(* --> Controller Errors <--*)
		17664	:		FC_NcErrorMsg:='Controller Errors-Parameter:"Controller ID not allowed" The value for the controller ID is not allowed,  e.g. because it has already been assigned, is less than or equal to zero, or is greater than 255.';
		17665	:		FC_NcErrorMsg:='Controller Errors-Parameter:"Controller type not allowed" The value for the controller type is unacceptable because it is not defined. Type 1: P-controller (position) . . .  Type 7: High/low speed controller  Type 8: JogStepper motor controller  Type 9: Sercos controller';
		17666	:		FC_NcErrorMsg:='Controller Errors-Parameter:"Controller operating mode not allowed" The value for the controller operating mode is not allowed.';
		17667	:		FC_NcErrorMsg:='Controller Errors-Parameter:"Weighting of the velocity pre-control not allowed" The value for the percentage weighting of the velocity pre-control is not allowed.  The parameter is pre-set to 1.0 (100%) as standard.';
		17668	:		FC_NcErrorMsg:='Controller Errors-Parameter:"Following error monitoring (position) not allowed" The value for the activation of the following error monitoring is not allowed.';
		17669	:		FC_NcErrorMsg:='Controller Errors-Parameter:"Following error (velocity) not allowed" The value for the activation of the following error monitoring (velocity) is not allowed.';
		17670	:		FC_NcErrorMsg:='Controller Errors-Parameter:"Following error window (position) not allowed" The value for the following error window (maximum allowable following error) is not allowed.';
		17671	:		FC_NcErrorMsg:='Controller Errors-Parameter:"Following error filter time (position) not allowed" The value for the following error filter time (position) is not allowed.';
		17672	:		FC_NcErrorMsg:='Controller Errors-Parameter:"Following error window (velocity) not allowed" The value for the following error window (velocity) is not allowed.';
		17673	:		FC_NcErrorMsg:='Controller Errors-Parameter:"Following error filter time (velocity) not allowed" The value for the following error filter time (velocity) is not allowed.';
		17680	:		FC_NcErrorMsg:='Controller Errors-Parameter:"Proportional gain Kv or Kp (position controller) not allowed" The value for the proportional gain (Kv factor or Kp factor) is not allowed.';
		17681	:		FC_NcErrorMsg:='Controller Errors-Parameter:"Integral-action time Tn (position controller) not allowed" The value for the integral-action time is not allowed (I proportion of the PID T1 controller).';
		17682	:		FC_NcErrorMsg:='Controller Errors-Parameter:"Derivative action time Tv (position controller) not allowed" The value for the derivative action time is not allowed (D proportion of the PID T1 controller).	';
		17683	:		FC_NcErrorMsg:='Controller Errors-Parameter:"Damping time Td (position controller) not allowed" The value for the damping time is not allowed (D proportion of the PID T1 controller).  Suggested value: 0.1 * Tv';
		17684	:		FC_NcErrorMsg:='Controller Errors-Function:"Activation of the automatic offset compensation not allowed" Activation of the automatic offset compensation is only possible for certain types of controller (with no I component).';
		17685	:		FC_NcErrorMsg:='Controller Errors-Parameter:"Additional proportional gain Kv or Kp (position controller) not allowed" The value for the second term of the proportional gain (Kv factor or Kp factor) is not allowed.';
		17686	:		FC_NcErrorMsg:='Controller Errors-Parameter:"Reference velocity for additional proportional gain Kv or Kp (position controller) not allowed"  The value for the reference velocity percentage data entry, to which the additional proportional gain is applied, is not allowed.  The standard setting for the parameter is 0.5 (50%).';
		17687	:		FC_NcErrorMsg:='Controller Errors-Parameter:"Proportional gain Pa (acceleration proportion) not allowed" The value for the proportional gain (Pa factor) is not allowed.	';
		17688	:		FC_NcErrorMsg:='Controller Errors-Parameter:"Proportional gain Kv (velocity controller) not allowed" The value for the proportional gain (Kv factor) is not allowed.';
		17689	:		FC_NcErrorMsg:='Controller Errors-Parameter:"Reset time Tn (velocity controller) not allowed” The value for the integral-action time is not allowed (I proportion of the PID T1 controller).';
		17690	:		FC_NcErrorMsg:='Controller Errors-Address:"CONTROLERR_RANGE_ACCJUMPLIMITINGMODE"';
		17691	:		FC_NcErrorMsg:='Controller Errors-Address:"CONTROLERR_RANGE_ACCJUMPVALUE"	';
		17692	:		FC_NcErrorMsg:='Controller Errors-Address:"CONTROLERR_RANGE_FILTERTIME"	';
		17693	:		FC_NcErrorMsg:='Controller Errors-Parameter:"Dead zone not allowed" The value for the dead zone from the position error or the velocity error (system deviation) is not allowed  (only for complex controller with velocity or torque interface).';
		17696	:		FC_NcErrorMsg:='Controller Errors-Parameter:”Rate time Tv (velocity controller) not allowed” The value for the derivative action time is not allowed (D proportion of the PID T1 controller).';
		17697	:		FC_NcErrorMsg:='Controller Errors-Parameter:"Damping time Td (velocity controller) not allowed" The value for the damping time is not allowed (D proportion of the PID T1 controller). Suggested value: 0.1 * Tv';
		17698	:		FC_NcErrorMsg:='Controller Errors-Parameter:"CONTROLERR_RANGE_IOUTPUTLIMIT"	';
		17699	:		FC_NcErrorMsg:='Controller Errors-Parameter:"CONTROLERR_RANGE_DOUTPUTLIMIT"	';
		17700	:		FC_NcErrorMsg:='Controller Errors-Parameter:"CONTROLERR_RANGE_POSIDISABLEWHENMOVING"	';
		17728	:		FC_NcErrorMsg:='Controller Errors-Initialization:"Controller initialisation" Controller has not been initialised. Although the controller has been created, the rest of the initialisation has not been performed (1. Initialisation of controller, 2. Reset controller).';
		17729	:		FC_NcErrorMsg:='Controller Errors-Address:"Axis address" Controller does not know its axis, or the axis address has not been initialised.';
		17730	:		FC_NcErrorMsg:='Controller Errors-Address:"Drive address" Controller does not know its drive, or the drive address has not been initialised.';
		17744	:		FC_NcErrorMsg:='Controller Errors-Monitoring:"Following error monitoring (position)" With active following error monitoring (position) a following error exceedance has occurred,  whose magnitude is greater than the following error window, and whose duration is longer than the parameterised following error filter time.';
		17745	:		FC_NcErrorMsg:='Controller Errors-Monitoring:"Following error monitoring (velocity)" With active following error monitoring (velocity) a velocity following error exceedance has occurred,  whose magnitude is greater than the following error window, and whose duration is longer than the parameterised following error filter time.';
		17824	:		FC_NcErrorMsg:='Controller Errors-Monitoring:"CONTROLERR_RANGE_AREA_ASIDE"';
		17825	:		FC_NcErrorMsg:='Controller Errors-Monitoring:"CONTROLERR_RANGE_AREA_BSIDE"';
		17826	:		FC_NcErrorMsg:='Controller Errors-Monitoring:"CONTROLERR_RANGE_QNENN"';
		17827	:		FC_NcErrorMsg:='Controller Errors-Monitoring:"CONTROLERR_RANGE_PNENN"';
		17828	:		FC_NcErrorMsg:='Controller Errors-Monitoring:"CONTROLERR_RANGE_AXISIDPRESP0"';


(* --> Drive Errors <--*)

		17920	:		FC_NcErrorMsg:='Drive Errors-Parameter:"Drive ID not allowed" The value for the drive ID is not allowed, e.g. because it has already been assigned, is less than or equal to zero, or is greater than 255.';
		17921	:		FC_NcErrorMsg:='Drive Errors-Parameter:"Drive type not allowed" The value for the drive type is unacceptable because it is not defined.';
		17922	:		FC_NcErrorMsg:='Drive Errors-Parameter:"Drive operating mode not allowed" The value for the drive operating mode is not allowed. Modus 1: Standard';
		17923	:		FC_NcErrorMsg:='Drive Errors-Parameter:"Motor polarity inverted?" The flag for the motor polarity is not allowed.  Flag 0: Positive motor polarity Flag 1: Negative motor polarity';
		17924	:		FC_NcErrorMsg:='Drive Errors-Parameter:"Drift compensation/velocity offset (DAC offset)" The value for the drift compensation (DAC offset) is not allowed.';
		17925	:		FC_NcErrorMsg:='Drive Errors-Parameter:"Reference velocity (velocity pre-control)" The value for the reference velocity (velocity pre-control) is not allowed.';
		17926	:		FC_NcErrorMsg:='Drive Errors-Parameter:"Reference output in percent" The value for the reference output in percent is not allowed.  The value 1.0 (100 %) usually corresponds to a voltage of 10.0 V.';
		17927	:		FC_NcErrorMsg:='Drive Errors-Parameter:"Quadrant compensation factor" The value for the quadrant compensation factor is not allowed.';
		17928	:		FC_NcErrorMsg:='Drive Errors-Parameter:"Velocity reference point in percent" The value for the velocity reference point in percent is not allowed. The value 1.0 corresponds to 100 percent.';
		17929	:		FC_NcErrorMsg:='Drive Errors-Parameter:"Output reference point in percent" The value for the output reference point in percent is not allowed. The value 1.0 corresponds to 100 percent.';
		17930	:		FC_NcErrorMsg:='Drive Errors-Parameter:"Minimum or maximum output limit" The values for the minimum and/or maximum output limit is not allowed. This will happen if the range of values is exceeded, The maximum limit is smaller than the minimum limit, or the distance between the minimum and maximum limits is zero. The minimum limit is initially set to 1.0 (-100 percent) and the maximum limit to 1.0 (100 percent).';
		17931	:		FC_NcErrorMsg:='Drive Errors-Parameter:"DRIVEERR_RANGE_MAXINCREMENT"';
		17932	:		FC_NcErrorMsg:='Drive Errors-Parameter:"DRIVEERR_RANGE_ DRIVECONTROLDWORD"';
		17933	:		FC_NcErrorMsg:='Drive Errors-Parameter:"DRIVEERR_RANGE_ RESETCYCLECOUNTER"';
		17935	:		FC_NcErrorMsg:='Drive Errors-Parameter:"Drive torque output scaling is not allowed" The value for the drive torque output scaling (rotary motor) or the force output scaling (linear motor) is not allowed.';
		17936	:		FC_NcErrorMsg:='Drive Errors-Parameter:"Drive velocity output scaling is not allowed" The value for the drive velocity output scaling is not allowed.';
		17937	:		FC_NcErrorMsg:='Drive Errors-Parameter:"Profi Drive DSC Proportional gain Kpc (position controller) not allowed" The value for the profi drive DSC proportional gain (Kpc factor) is not allowed.';
		17938	:		FC_NcErrorMsg:='Drive Errors-Parameter:"Table-ID is invalid" The value for the table-ID is invalid.';
		17939	:		FC_NcErrorMsg:='Drive Errors-Parameter:"Table interpolationtype is invalid" The value for the table interpolation-type is invalid.';
		17940	:		FC_NcErrorMsg:='Drive Errors-Parameter:"Outputoffset in percent is invalid" The value for the output offset in percent (+/- 1.0) is invalid.';
		17941	:		FC_NcErrorMsg:='Drive Errors-Parameter:"Profi Drive DSC scaling factor for calculating "Xerr" (position controller) is not allowed"  The value as profi drive DSC scaling factor for calculating "Xerr" is invalid.';
		17942	:		FC_NcErrorMsg:='Drive Errors-Parameter:"Drive acceleration output scaling is not allowed" The value for the drive acceleration/deceleration output scaling is not allowed.';
		17943	:		FC_NcErrorMsg:='Drive Errors-Parameter:"Drive position output scaling is not allowed" The value for the drive position output scaling is not allowed.';
		17952	:		FC_NcErrorMsg:='Drive Errors-Parameter:"Bit mask for JogStepper motor cycle not allowed" A value in the various JogStepper motor masks for the cycle concerned is not allowed.';
		17953	:		FC_NcErrorMsg:='Drive Errors-Parameter:"Bit mask for JogStepper motor holding current not allowed" The value for the JogStepper motor holding mask is not allowed.';

		17968	:		FC_NcErrorMsg:='Drive Errors-Monitoring:"Overtemperature" The drive resp. terminal detects an overtemperature alarm.';
		17969	:		FC_NcErrorMsg:='Drive Errors-Monitoring:"Undervoltage" The drive resp. terminal detects an undervoltage (supply voltage to low).	';
		17970	:		FC_NcErrorMsg:='Drive Errors-Monitoring:"Wire breakage in phase A" The drive resp. terminal detects a wire breakage in phase A.';
		17971	:		FC_NcErrorMsg:='Drive Errors-Monitoring:"Wire breakage in phase B" The drive resp. terminal detects a wire breakage in phase B.';
		17972	:		FC_NcErrorMsg:='Drive Errors-Monitoring:"Overcurrent in phase A" The drive resp. terminal detects an overcurrent in phase A.';
		17973	:		FC_NcErrorMsg:='Drive Errors-Monitoring:"Overcurrent in Phase B" The drive resp. terminal detects an overcurrent in phase B.	';
		17974	:		FC_NcErrorMsg:='Drive Errors-Monitoring:"Torque overload (stall situation)" The drive resp. terminal detects a torque overload (stall situation).';
		17984	:		FC_NcErrorMsg:='Drive Errors-Initialization:"Drive initialisation" Drive has not been initialised.  Although the drive has been created, the rest of the initialisation has not been performed  (1. Initialisation of drive I/O, 2. Initialisation of drive, 3. Reset drive).';
		17985	:		FC_NcErrorMsg:='Drive Errors-Address:"Axis address" Drive does not know its axis, or the axis address has not been initialised.';
		17986	:		FC_NcErrorMsg:='Drive Errors-Address:"I/O input structure address" The drive does not have a valid I/O input address in the process image.';
		17987	:		FC_NcErrorMsg:='Drive Errors-Address:"I/O output structure address" The drive does not have a valid I/O output address in the process image.';
		18000	:		FC_NcErrorMsg:='Drive Errors-Monitoring:"Drive not ready for operation" The drive is not ready for operation. The following are possible causes: - the drive is in failure state (hardware fault) - the drive is in the starting-up stage  (e.g. following an axis reset preceded by a hardware fault) - the drive has not been enabled Remark:  The time required for "booting" a drive after a hardware fault can amount to several seconds.	';
		18001	:		FC_NcErrorMsg:='Drive Errors-Monitoring:"Error in cyclic communication with the drive (life counter)", The reason for this could be an interruption in the fieldbus or that the drive is in an error state.';
		18002	:		FC_NcErrorMsg:='Drive Errors-Monitoring:"Not permitted to change the table ID while the axis is enabled",It is not permitted to change the table ID while the axis/drive is enabled.';
		18005	:		FC_NcErrorMsg:='Drive Errors-Monitoring:"Invalid IO data for more than "n" consecutive nc cycles",The axis (encoder or drive) detects for more than "n" consecutive nc cycles invalid IO data (e.g. n=3), As a result it is possible that the encoder calibration flag will set to FALSE (that means uncalibrated); EtherCAT field bus: working counter error ("WCState") ;  Lightbus field bus: CDL state error ("CdlState")';


(* --> NC-CAM Errors <--*)
		18944	:		FC_NcErrorMsg:='	Nc Cam Errors-	parameter:	"Table ID not allowed" The value for the table ID is not allowed, e.g. because it has already been assigned, is less than or equal to zero, or is greater than 255. 		';
		18945	:		FC_NcErrorMsg:='	Nc Cam Errors-	parameter	:	"Table type not allowed" The value for the table type is unacceptable because it is not defined. 		';
		18946	:		FC_NcErrorMsg:='	Nc Cam Errors-	parameter	:	"Number of lines in the table not allowed" The value of the number of lines in the table is not allowed, because for example, it is smaller than two at linear interpolation and smaller than four at spline interpolation. 		';
		18947	:		FC_NcErrorMsg:='	Nc Cam Errors-	parameter	:	"Number of columns in the table is not allowed" The value of the number of columns in the table is not allowed, because for example, it is less than or equal to zero (depends upon the type of table or slave). 		';
		18948	:		FC_NcErrorMsg:='	Nc Cam Errors-	parameter	:	"JogStep size (position delta) not allowed" The value for the JogStep size between two lines (position delta) is not allowed, because for example, it is less than or equal to zero. 		';
		18949	:		FC_NcErrorMsg:='	Nc Cam Errors-	parameter	:	"Period not allowed" The value for the period is not allowed, because for example, it is less than or equal to zero. 		';
		18950	:		FC_NcErrorMsg:='	Nc Cam Errors-	parameter	:	"Table is not monotonic" The value for the JogStep size is not allowed, because for example, it is less than or equal to zero.		';
		18951	:		FC_NcErrorMsg:='	Nc Cam Errors-	initialization	:	„Table sub type is not allowed” The value for the table sub type is not allowed or otherwise the table class (slave type) do not match up to the table main type.$NTable sub type: (1) equidistant linear position table, (2) equidistant cyclic position table, (3) none equidistant linear position table, (4) none equidistant cyclic position table		';
		18952	:		FC_NcErrorMsg:='	Nc Cam Errors-	initialization	:	„Table interpolation type is not allowed” The value for the table interpolation type is allowed$NTable interpolation type: (0) linear-interpolation, (1) 4-point-interpolation, (2) spline-interpolation		';
		18953	:		FC_NcErrorMsg:='	Nc Cam Errors-	initialization	:	"Incorrect table main type" The table main type is unknown or otherwise the table class (slave type) do not match up to the table main type.$NTable main type: (1) camming table, (2) characteristic table, (3) motion FUNCTION table (MF)		';
		18960	:		FC_NcErrorMsg:='	Nc Cam Errors-	initialization	:	"Table initialisation" Table has not been initialised. Although the table has been created, the rest of the initialisation has not been performed. For instance, the number of lines or columns may be less than or equal to zero.	';
		18961	:		FC_NcErrorMsg:='	Nc Cam Errors-	initialization	:	"Not enough memory" Table could not be created, since there is not enough memory.		';
		18962	:		FC_NcErrorMsg:='	Nc Cam Errors-	function	:	"Function not executed, function not available" The function has not been implemented, or cannot be executed, for the present type of table.		';
		18963	:		FC_NcErrorMsg:='	Nc Cam Errors-	function	:	"Line index not allowed" The start line index or the stop line index to be used for read or write access to the table is not allowed. $NFor instance, the line index may be greater than the total number of lines in the table.		';
		18964	:		FC_NcErrorMsg:='	Nc Cam Errors-	function	:	"Column index not allowed" The start column index or the stop column index to be used for read or write access to the table in not allowed. For instance, the column index may be greater than the total number of columns in the table.		';
		18965	:		FC_NcErrorMsg:='	Nc Cam Errors-	function	:	"Number of lines not allowed" The number of lines to be read from or written to the table is not allowed. $NThe number of lines must be an integer multiple of the number of elements in a line (n * number of columns).		';
		18966	:		FC_NcErrorMsg:='	Nc Cam Errors-	function	:	"Number of columns not allowed" The number of columns to be read from or written to the table is not allowed.$NThe number of columns must be an integer multiple of the number of elements in a column (n * number of lines).  		';
		18967	:		FC_NcErrorMsg:='	Nc Cam Errors-	function	:	"Error in scaling or in range entry" The entries in the table header are inconsistent, e.g. the validity range is empty. $NIf the error is generated during the run time it is a run time error and stops the master/slave group.		';
		18968	:		FC_NcErrorMsg:='	Nc Cam Errors-	function	:	"Multi table slave out of range" The slave master position is outside the table values for the master. The error is a run-time error, and stops the master/slave group.		';
		18969	:		FC_NcErrorMsg:='	Nc Cam Errors-	function	:	"Solo table underflow" The slave master position is outside the table values for the master. The master value of the equidistant table, to be processed linearly, lies under the first table value. $NThe error is a run-time error, and stops the master/slave group.		';
		18970	:		FC_NcErrorMsg:='	Nc Cam Errors-	function	:	"Solo table overflow" The slave master position is outside the table values for the master. The master value of the equidistant table, to be processed linearly, lies above the first table value. $NThe error is a run-time error, and stops the master/slave group.		';
		18971	:		FC_NcErrorMsg:='	Nc Cam Errors-	parameter	:	"Incorrect execution mode" The cyclic execution mode can only be "true" or "false".		';
		18972	:		FC_NcErrorMsg:='	Nc Cam Errors-	parameter	:	"Impermissible parameter" The Fifo parameter is not allowed.		';
		18973	:		FC_NcErrorMsg:='	Nc Cam Errors-	parameter	:	"Fifo is empty" The Fifo of the external generator is empty. This can signify end of track or a run time error.		';
		18974	:		FC_NcErrorMsg:='	Nc Cam Errors-	parameter	:	"Fifo is full" The Fifo of the external generator is full. It is the user‘s task to continue to attempt to fill the Fifo with the rejected values.		';
		18975	:		FC_NcErrorMsg:='	Nc Cam Errors-	parameter	:	„Point-Index of Motion Function invalid”  The point index of a Motion Function Point of a Function Table is invalid. $NFirst the point index has to be larger than zero and second it has to be numerical continuously for one column in the Montion Function Table (e.g. 1,2,3,... or 10,11,12,...).$NnRemark: The point index is not online-changeable but must be constant.		';
		18976	:		FC_NcErrorMsg:='	Nc Cam Errors-	initialization	:	„No diagonalisation of  matrix” The spline can not be calculated. The master positions are not correct.		';
		18977	:		FC_NcErrorMsg:='	Nc Cam Errors-	initialization	:	„Number of spline points to less” The number of points of a cubic spline has to be greater than two.		';
		18978	:		FC_NcErrorMsg:='	Nc Cam Errors-	initialization	:	„Fifo must not be overwritten” Fifo must not be overwritten since then the active line would be overwritten. $NIt is the task of the user to secure that the active line is not modified.		';


(* --> NC-PLC Errors <--*)

		19200	:		FC_NcErrorMsg:='NC-PLC Errors-Parameter:"Axis has been stopped" The axis has been stopped while the axis moves to target position.  The axis could be stopped with a PLC Command via ADS, with the call of AXFNC or with the TwinCAT System Manager.';
		19201	:		FC_NcErrorMsg:='NC-PLC Errors-Parameter:"Axis cannot be started" The axis cannot be started, because: the axis is in an error state, the axis is doing another job,  The axis in protected mode, the axis is not in a ready state.';
		19202	:		FC_NcErrorMsg:='NC-PLC Errors-Parameter:"Control mode not allowed" No Target Position Control and no Position Area Control.';
		19203	:		FC_NcErrorMsg:='NC-PLC Errors-Parameter:"Axis is not moving" Restart position and velocity is only allowed if axis is physically moving.';
		19204	:		FC_NcErrorMsg:='NC-PLC Errors-Parameter:"Wrong mode for RestartPosAndVelo" Wrong mode.';
		19205	:		FC_NcErrorMsg:='NC-PLC Errors-Parameter:"Command not allowed": Endless move to a non specified direction;Read/Write parameter: type mismatch';
		19206	:		FC_NcErrorMsg:='NC-PLC Errors-Parameter:"Parameter not correct"	:Wrong override: > 100% or < 0%	;Wrong gearing factor: RatioDenominator = 0	;Wrong register into process (Register communication)';
		19207	:		FC_NcErrorMsg:='NC-PLC Errors-Parameter:"Timeout axis function block":After positioning, all "MC_Move..." blocks check whether positioning was completed successfully. In the simplest case, the "AxisHasJob" flag of the NC axis is checked, which initially signifies that positioning was logically completed. Depending on the parameterisation of the NC axis,  further checks (quality criteria) are used:"Position range monitoring"	If position range monitoring is active,  the system waits for feedback from the NC.  After positioning, the axis must be within the specified positioning range window. If necessary, the position controller ensures that the axis is moved to the target position.  If the position controller is switched off (Kv=0) or weak, the target may not be reached."Target position monitoring" If target position monitoring is active, the system waits for feedback from the NC.  After positioning, the axis must be within the specified target position window for at least the specified time.  If necessary, the position controller ensures that the axis is moved to the target position.  If the position controller is switched off (Kv=0) or weak, the target may not be reached.  Floating position control may lead to the axis oscillating around the window but not remaining inside the window. If the axis is logically at the target position (logical standstill) but the parameterised position window has not been reached,  monitoring of the above-mentioned NC feedback is aborted with error 19207 (0x4B07) after a constant timeout of 6 seconds. ';
		19208	:		FC_NcErrorMsg:='NC-PLC Errors-Parameter:"Axis in protected mode" Axis is in protected mode (i.e. coupled) and cannot be moved.';
		19209	:		FC_NcErrorMsg:='NC-PLC Errors-Parameter:"Axis is not ready" Axis is not ready and cannot be moved.';
		19210	:		FC_NcErrorMsg:='NC-PLC Errors-Parameter:"Homing error" The Homing of an axis could not be started or was not successful';
		19211	:		FC_NcErrorMsg:='NC-PLC Errors-Parameter:"Invalid definition trigger input definition" The definition of the trigger signal used with the function block MC_TouchProbe is invalid.  The defined encoder ID, the trigger signal or the trigger signal edge are invalid.';
		19212	:		FC_NcErrorMsg:='NC-PLC Errors-Function:"position latch has been deactivated" The function block MC_TouchProbe encountered that a touch probe sequence has been deactivated after the block started this sequence.  The reason for instance can be an axis reset.';
		19213	:		FC_NcErrorMsg:='NC-PLC Errors-Function:"Timeout NC status feedback" A function block has successfully executed a command but the NC does not pass the expected feedback in the axis status word.';
		19214	:		FC_NcErrorMsg:='NC-PLC Errors-Function:"Supplement not installed" - The function is available as supplement product but not installed on the system.';
		19215	:		FC_NcErrorMsg:='NC-PLC Errors-Function:"Timeout Register Access" - The access to a bus terminal register timed out.';
		19216	:		FC_NcErrorMsg:='NC-PLC Errors-Function:"M-Function request missing" This error occurs if a confirmation of an M-Function is made but the request bit is not set.';
		19217	:		FC_NcErrorMsg:='NC-PLC Errors-Parameter:"Zero shift index is out of range" The index of the zero shift is invalid';
		19218	:		FC_NcErrorMsg:='NC-PLC Errors-Parameter:"R parameter index or size is invalid". This error occurs, if the R parameters are written or read and the index or size is out of range';
		19219	:		FC_NcErrorMsg:='NC-PLC Errors-Parameter:"Index for tool description is invalid"';
		19220	:		FC_NcErrorMsg:='NC-PLC Errors-Function:"Version of cyclic channel interface does not match to the requested function and function block, resp."  This error occurs, if an older TwinCAT Version is used and a new functionality from a newer TcNci.lib is called.';
		19221	:		FC_NcErrorMsg:='NC-PLC Errors-Function:"Channel is not ready for requested function". The requested function can not be executed due to a wrong state of the channel.  This error occurs for instance, if retrace is requested and the axes are not stopped with ItpEStop before.';
		19222	:		FC_NcErrorMsg:='NC-PLC Errors-Function:"Requested function is not turned on". The requested function requires an explicit activation before it can be executed.';
		19232	:		FC_NcErrorMsg:='NC-PLC Errors-Parameter:"Cannot append all axes". This error occurs, if you want to append an auxiliary axes to an interpolation group and the function fails.  Probably a prior assignment of an auxiliary axes was skipped.';
		19248	:		FC_NcErrorMsg:='NC-PLC Errors-Parameter:"Pointer invalid". The pointer to a data structure is invalid, e.g. NULL.:data structure MC_CAM_REF is possibly not initialized';
		19249	:		FC_NcErrorMsg:='NC-PLC Errors-Parameter:"Size of memory invalid". The size parameter is invalid:The value of the size parameter is 0 or less than the size of one element of the addressed data structure. The value of the size parameter is less than the requested amount of data. The value of the size parameter does not match other parameters as number of points, number of rows or number of columns.';
		19250	:		FC_NcErrorMsg:='NC-PLC Errors-Parameter:"Invalid cam table ID". The cam table ID is out of the range from 1 to 255.';
		19251	:		FC_NcErrorMsg:='NC-PLC Errors-Parameter:"Invalid point ID". The point ID of a motion function point is lower than 1.';
		19252	:		FC_NcErrorMsg:='NC-PLC Errors-Parameter:"Invalid number of points ". The number of points to read or write is less than 1.';
		19253	:		FC_NcErrorMsg:='NC-PLC Errors-Parameter:"Invalid MC table type". The type of a cam table does not match the MC_TableType definition.';
		19254	:		FC_NcErrorMsg:='NC-PLC Errors-Parameter:"Invalid number of rows". The number of rows of a cam table is less than 1.';
		19255	:		FC_NcErrorMsg:='NC-PLC Errors-Parameter:"Invalid number of columns". The number of columns of a cam table is invalid. The number of columns of a motion function is not equal to 1 ;The number of columns of a standard cam table is not equal to 2 The number of columns does not match other parameters (ValueSelectMask)';
		19256	:		FC_NcErrorMsg:='NC-PLC Errors-Parameter:"Invalid Increment". The increment for an interpolation is invalid, e.g. <= 0.';
		19264	:		FC_NcErrorMsg:='NC-PLC Errors-Monitoring:"Unsupported Terminal Type". The terminal in use is not supported by this function block.';
		19265	:		FC_NcErrorMsg:='NC-PLC Errors-Monitoring:"Register Read/Write Error". This error implies to be a validation error.';
		19266	:		FC_NcErrorMsg:='NC-PLC Errors-Monitoring:"Axis is Enabled". Axis is enabled and is not supposed to be enabled for this operation';
		19267	:		FC_NcErrorMsg:='NC-PLC Errors-Parameter:"Size of compensation table wrong". The stated table size in bytes is not conform with the real size.';
		19268	:		FC_NcErrorMsg:='NC-PLC Errors-Parameter:The minimum/ maximum position of the compenstation table is not conform to the position in the table description (ST_CompensationDesc)';
		19269	:		FC_NcErrorMsg:='NC-PLC Errors-Parameter:"Not implemented". The requested function is not implemented in this combination.';
		19296	:		FC_NcErrorMsg:='NC-PLC Errors-Monitoring:"Motion command not be activated". A motion command has been started and has been buffered and confirmed by the NC. Nevertheless the command did not become active.';
		19297	:		FC_NcErrorMsg:='NC-PLC Errors-Monitoring:"Motion command could not be monitored by the PLC". A motion command has been started and has been buffered and confirmed by the NC.  The PLC has not been able to monitor the execution of this command and the execution status is unclear since the NC is already executing a more recent command.  This error may com up with very short buffered motion commands which are executed during one PLC cycle.';
		19298	:		FC_NcErrorMsg:='NC-PLC Errors-Monitoring:"Buffered command finished with error". A buffered command finished with an error. The error number is not available because a new command is already in execution.';
		19299	:		FC_NcErrorMsg:='NC-PLC Errors-Monitoring:"Buffered command finished without state feedback". A buffered command finished without success or error feedback.';
		19300	:		FC_NcErrorMsg:='NC-PLC Errors-Monitoring:" "BufferMode" not supported". The "BufferMode" is not supported by the command.';
		19301	:		FC_NcErrorMsg:='NC-PLC Errors-Monitoring:"Command number is zero". The system administrated command number for buffered commands is zero.';
		19313	:		FC_NcErrorMsg:='NC-PLC Errors-Parameter:"Invalid NCI Entry Type". FB_NciFeedTablePreparation is called with an unknown nEntryType';
		19314	:		FC_NcErrorMsg:='NC-PLC Errors-Function:"NciFeedTable full". The table is full filled and therefore this entry is not accepted. To do:Transfer the context of the table with FB_NciFeedTable to the NC-Kernel.  If this succeeded bFeedingDone becomes TRUE and the context of the table has to be reset with bResetTable (FB_NciFeedTablePreparation).  Now the table can be refilled with new entries.';
		19315	:		FC_NcErrorMsg:='NC-PLC Errors-Function:internal error';
		19316	:		FC_NcErrorMsg:='NC-PLC Errors-Parameter:$NST_NciTangentialFollowingDesc: tangential axis is not an auxiliary axis"  The entry ST_NciTangentialFollowingDesc contains an tangential axis that is no auxiliary axis.';
		19317	:		FC_NcErrorMsg:='NC-PLC Errors-Parameter:$NST_NciTangentialFollowingDesc: nPathAxis1 and nPathAxis2, resp. are no path axes. So it is not possible to determine the plane.';
		19318	:		FC_NcErrorMsg:='NC-PLC Errors-Parameter:$NST_NciTangentialFollwoingDesc: nPathAxis1 and nPathAxis2 are equal. So it is not possible to determine the plane.';
		19319	:		FC_NcErrorMsg:='NC-PLC Errors-Parameter:$NST_NciGeoCirclePlane: circle is programmed in a wrong manner.';
		19320	:		FC_NcErrorMsg:='NC-PLC Errors-Function:$NInternal error in calculation of the tangential following';
		19321	:		FC_NcErrorMsg:='NC-PLC Errors-Monitoring:$NTangential following: With ST_NciTangentialFollowingDesc the monitoring of the deviation angle (E_TfErrorOnCrirical1)  is activated and with the actual segment the deviation angle is too big.';
		19322	:		FC_NcErrorMsg:='NC-PLC Errors-Function:$Nnot implemented';
		19323	:		FC_NcErrorMsg:='NC-PLC Errors-Parameter:$NTangential Following: The radius of the actual circle segment is too small';
		19324	:		FC_NcErrorMsg:='NC-PLC Errors-Parameter:$NFB_NciFeedTablePreparation: pEntry is NULL';
		19325	:		FC_NcErrorMsg:='NC-PLC Errors-Parameter:$NFB_NciFeedTablePreparation: The specified nEntryType does not match the the structure type';
		19326	:		FC_NcErrorMsg:='NC-PLC Errors-Parameter:$NST_NciMFuncFast and ST_NciMFuncHsk: The requested m-function is not in between 0..159';
		19327	:		FC_NcErrorMsg:='NC-PLC Errors-Parameter:$NST_NciDynOvr: The requested value for the dynamic override is not in between 0.01 and 1.0';
		19328	:		FC_NcErrorMsg:='NC-PLC Errors-Parameter:$NST_NciVertexSmoothing: invalid parameter. This error occurs with a negative vertex radius or an unknown vertex smoothing type.';
		19329	:		FC_NcErrorMsg:='NC-PLC Errors-Parameter:$NFB_NciFeedTablePrepartion: The requested velocity is not in a valid range';
		19330	:		FC_NcErrorMsg:='NC-PLC Errors-Parameter:$NST_Nci*: invalid parameter';



		33056	:	FC_NcErrorMsg:='NC3_Environment_Invalid configuration for Object (e.g. in System Manager)';
		33057	:	FC_NcErrorMsg:='NC3_Environment_Invalid environment FOR Object (e.g. TcCom-Object Hierarchy OR missing/faulty Objects)';
		33058	:	FC_NcErrorMsg:='NC3_Environment_Incompatible Driver OR Object';
		33084	:	FC_NcErrorMsg:='NC3_Parameter_BufferMode is invalid';
		33085	:	FC_NcErrorMsg:='NC3_FunctionBlock_Only one active Instance OF FUNCTION Block per Group is allowed';
		33086	:	FC_NcErrorMsg:='NC3_State_Command is NOT allowed in current group state';
		33087	:	FC_NcErrorMsg:='NC3_FunctionBlock_Slave cannot synchronize.The slave cannot reach the SlaveSyncPosition BY the TIME the master has reached the MasterSyncPos';
		33088	:	FC_NcErrorMsg:='NC3_Parameter_Invalid value FOR one OR more OF the dynamic parameters (A, D, J)';
		33089	:	FC_NcErrorMsg:='NC3_Parameter_IdentInGroup is invalid';
		33090	:	FC_NcErrorMsg:='NC3_Parameter_The number OF axes in the group is incompatible with the axes convention';
		33091	:	FC_NcErrorMsg:='NC3_Communication_FUNCTION Block OR respective Command is NOT supported BY Target';
		33093	:	FC_NcErrorMsg:='NC3_FunctionBlock_Mapping OF Cyclic INTERFACE between Nc AND Plc missing (e.g. AXIS_REF, AXES_GROUP_REF, ...)';
		33094	:	FC_NcErrorMsg:='NC3_FunctionBlock_Invalid Velocity ValueThe velocity was NOT set OR the entered value is invalid';
		33096	:	FC_NcErrorMsg:='NC3_FunctionBlock_Invalid Input Value';
		33097	:	FC_NcErrorMsg:='NC3_FunctionBlock_Invalid OR Incomplete Input ARRAY';
		33098	:	FC_NcErrorMsg:='NC3_Parameter_Unsupported Dynamics FOR selected Group Kernel';
			
		
		ELSE
			IF 36844<error AND error< 36857 THEN
				FC_NcErrorMsg:='NC3_Internal_Unexpected INTERNAL Error';
			ELSE		
				FC_NcErrorMsg:='Msg Unknown';
			END_IF	
END_CASE

END_FUNCTION

(* stored: Version 1.1.0.1, ProductVersion 3.1.4024.3
   POU FC_NcErrorMsg: Id {2cdd0c23-f932-04e5-1f15-c2f1cd63285a}, SpecialFunc None *)
